(* IEC 61131-3 sources: com.logicals.lc3.examples/TF_Training/src/Blocks/Motor/FBD, 3 files *)

(* ---- FB_Motor1D_FBD.iecfbd ---- *)
FUNCTION_BLOCK FB_Motor1D_FBD
  VAR
    FB_MotorRS : RS;
    FB_MotorR_TRIG : R_TRIG;
    FB_MotorTON : TON;
  END_VAR
  VAR_INPUT
    vix_Start : BOOL;
    vix_Stop : BOOL;
  END_VAR
  VAR_OUTPUT
    vox_MotorOut : BOOL;
    vox_Err : BOOL;
    vox_ErrNo : INT;
  END_VAR

  (*

    // Network 1:
    FB_MotorR_TRIG(CLK := vix_Start);
    FB_MotorRS(S := FB_MotorR_TRIG.Q, R1 := vix_Stop, Q1 => vox_MotorOut);

    // Network 2:
    AND(IN1 := vix_Start, IN2 := vix_Stop, AND => vox_Err);

    // Network 3:
    AND(IN1 := vix_Start, IN2 := vix_Stop, AND => @C(19).AND);
    MOVE(EN := @C(19).AND, IN := 1, MOVE => vox_ErrNo);

  *)

  @CF(11) : @R(620.0, 130.0, 670.0, 39.0), @T("Motor_1D"), @POU;
  @VF(1) : @E(vix_Start), @R(620.0, 210.0, 140.0, 19.0);
  @VF(2) : @E(vix_Stop), @R(620.0, 260.0, 140.0, 19.0);
  @C(3) : @FB(FB_MotorR_TRIG), @R(840.0, 210.0, 140.0, 18.0), @I(@N(CLK), @L(9.5)), @O(@N(Q), @R(9.5));
  @C(4) : @FB(FB_MotorRS), @R(1030.0, 210.0, 80.0, 38.0), @I(@N(S), @L(9.5)), @I(@N(R1), @L(29.5)), @O(@N(Q1), @R(9.5));
  @VF(8) : @E(vox_MotorOut), @R(1150.0, 210.0, 140.0, 19.0);
  @CF(10) : @R(620.0, 330.0, 670.0, 39.0), @T("Motor_1D - Error Bit"), @POU;
  @VF(12) : @E(vix_Start), @R(620.0, 400.0, 140.0, 19.0);
  @VF(13) : @E(vix_Stop), @R(620.0, 420.0, 140.0, 19.0);
  @C(14) : @F(AND), @R(860.0, 400.0, 40.0, 38.0), BOOL, @I(@N(IN1), @L(9.5)), @I(@N(IN2), @L(29.5)), @O(@N(AND), @R(9.5));
  @VF(17) : @E(vox_Err), @R(1150.0, 400.0, 140.0, 19.0);
  @C(19) : @F(AND), @R(860.0, 560.0, 40.0, 38.0), BOOL, @I(@N(IN1), @L(9.5)), @I(@N(IN2), @L(29.5)), @O(@N(AND), @R(9.5));
  @VF(20) : @E(vix_Start), @R(620.0, 560.0, 140.0, 19.0);
  @VF(21) : @E(vix_Stop), @R(620.0, 580.0, 140.0, 19.0);
  @VF(22) : @E(vox_ErrNo), @R(1150.0, 580.0, 140.0, 19.0);
  @CF(23) : @R(620.0, 490.0, 670.0, 39.0), @T("Motor_1D - Error No"), @POU;
  @C(26) : @F(MOVE), @R(1000.0, 560.0, 60.0, 38.0), INT, @I(@N(EN), @L(9.5)), @I(@N(IN), @L(29.5)), @O(@N(ENO), @R(9.5)), @O(@N(MOVE), @R(29.5));
  @VF(29) : @E(1), @R(760.0, 620.0, 140.0, 19.0), INT;
  @OLT(31) : @R(1360.0, 210.0, 80.0, 19.0), @S(8);

  @G(5) :
     @L(@VF(1).o, @C(3).CLK)
    ;
  @G(6) :
     @L(@C(3).Q, @C(4).S)
    ;
  @G(7) :
     @L(@VF(2).o, @C(4).R1)
    ;
  @G(9) :
     @L(@C(4).Q1, @VF(8).i)
    ;
  @G(15) :
     @L(@VF(12).o, @C(14).IN1)
    ;
  @G(16) :
     @L(@VF(13).o, @C(14).IN2)
    ;
  @G(18) :
     @L(@C(14).AND, @VF(17).i)
    ;
  @G(24) :
     @L(@VF(20).o, @C(19).IN1)
    ;
  @G(25) :
     @L(@VF(21).o, @C(19).IN2)
    ;
  @G(27) :
     @L(@C(19).AND, @C(26).EN)
    ;
  @G(28) :
     @L(@C(26).MOVE, @VF(22).i)
    ;
  @G(30) :
     @L(@VF(29).o, @C(26).IN)
    ;
END_FUNCTION_BLOCK

(* ---- FB_Motor2D_FBD.iecfbd ---- *)
FUNCTION_BLOCK FB_Motor2D_FBD
  {
    width := 310;
  }

  VAR
    FB_LeftRS : RS;
    FB_RightRS : RS;
    FB_LeftR_TRIG : R_TRIG;
    FB_RightR_TRIG : R_TRIG;
    FB_LeftTON : TON;
    FB_RightTON : TON;
  END_VAR
  VAR
    lx_LeftPulse : BOOL;
    lx_RightPulse : BOOL;
  END_VAR
  VAR_INPUT
    vix_Left : BOOL;
    vix_Right : BOOL;
    vix_LeftFB : BOOL;
    vix_RightFB : BOOL;
    vit_LeftFBTime : TIME := T#10m;
    vit_RightFBTime : TIME := T#10m;
  END_VAR
  VAR_OUTPUT
    vox_MotorLeft : BOOL;
    vox_MotorRight : BOOL;
    vox_LeftFBErr : BOOL;
    vox_RightFBErr : BOOL;
    vox_Err : BOOL;
    vox_ErrNo : INT;
  END_VAR

  (*

    // Network 1:
    FB_RightR_TRIG(CLK := vix_Right, Q => lx_RightPulse);

    // Network 2:
    FB_LeftR_TRIG(CLK := vix_Left, Q => lx_LeftPulse);

    // Network 3:
    AND(IN1 := vix_Left, IN2 := vix_Right, AND => vox_Err);

    // Network 4:
    AND(IN1 := vix_Left, IN2 := vix_Right, AND => @C(39).AND);
    MOVE(EN := @C(39).AND, IN := 1, MOVE => vox_ErrNo);

    // Network 5:
    FB_RightRS(S := lx_RightPulse, R1 := vox_MotorLeft, Q1 => vox_MotorRight);

    // Network 6:
    FB_LeftRS(S := lx_LeftPulse, R1 := vox_MotorRight, Q1 => vox_MotorLeft);

  *)

  @C(1) : @FB(FB_RightR_TRIG), @R(910.0, 150.0, 140.0, 18.0), @I(@N(CLK), @L(9.5)), @O(@N(Q), @R(9.5));
  @C(2) : @FB(FB_LeftR_TRIG), @R(910.0, 250.0, 140.0, 18.0), @I(@N(CLK), @L(9.5)), @O(@N(Q), @R(9.5));
  @VF(3) : @E(lx_LeftPulse), @R(1180.0, 250.0, 140.0, 19.0);
  @VF(4) : @E(lx_RightPulse), @R(1180.0, 150.0, 140.0, 19.0);
  @VF(7) : @E(vix_Left), @R(650.0, 250.0, 140.0, 19.0);
  @VF(9) : @E(vix_Right), @R(650.0, 150.0, 140.0, 19.0);
  @CF(11) : @R(650.0, 90.0, 670.0, 39.0), @T("Right R_TRIG"), @POU;
  @CF(12) : @R(650.0, 190.0, 670.0, 39.0), @T("Left R_TRIG"), @POU;
  @C(13) : @FB(FB_LeftRS), @R(990.0, 520.0, 80.0, 38.0), @I(@N(S), @L(9.5)), @I(@N(R1), @L(29.5)), @O(@N(Q1), @R(9.5));
  @C(14) : @FB(FB_RightRS), @R(990.0, 400.0, 80.0, 38.0), @I(@N(S), @L(9.5)), @I(@N(R1), @L(29.5)), @O(@N(Q1), @R(9.5));
  @VF(15) : @E(lx_RightPulse), @R(650.0, 400.0, 140.0, 19.0);
  @VF(17) : @E(lx_LeftPulse), @R(650.0, 520.0, 140.0, 19.0);
  @VF(19) : @E(vox_MotorLeft), @R(1180.0, 520.0, 140.0, 19.0);
  @VF(21) : @E(vox_MotorRight), @R(1180.0, 400.0, 140.0, 19.0);
  @CF(23) : @R(650.0, 330.0, 670.0, 39.0), @T("Left turn"), @POU;
  @CF(24) : @R(650.0, 460.0, 670.0, 39.0), @T("Right turn"), @POU;
  @VF(25) : @E(vox_MotorLeft), @R(650.0, 420.0, 140.0, 19.0);
  @VF(27) : @E(vox_MotorRight), @R(650.0, 540.0, 140.0, 19.0);
  @CF(29) : @R(650.0, 640.0, 680.0, 39.0), @T("Error bit"), @POU;
  @VF(30) : @E(vox_Err), @R(1190.0, 700.0, 140.0, 19.0);
  @VF(31) : @E(vix_Left), @R(660.0, 700.0, 140.0, 19.0);
  @VF(32) : @E(vix_Right), @R(660.0, 720.0, 140.0, 19.0);
  @C(33) : @F(AND), @R(1000.0, 700.0, 40.0, 38.0), BOOL, @I(@N(IN1), @L(9.5)), @I(@N(IN2), @L(29.5)), @O(@N(AND), @R(9.5));
  @CF(37) : @R(650.0, 780.0, 680.0, 39.0), @T("Error no"), @POU;
  @VF(38) : @E(vox_ErrNo), @R(1190.0, 880.0, 140.0, 19.0);
  @C(39) : @F(AND), @R(970.0, 860.0, 40.0, 38.0), BOOL, @I(@N(IN1), @L(9.5)), @I(@N(IN2), @L(29.5)), @O(@N(AND), @R(9.5));
  @VF(40) : @E(vix_Left), @R(660.0, 860.0, 140.0, 19.0);
  @VF(41) : @E(vix_Right), @R(660.0, 880.0, 140.0, 19.0);
  @C(44) : @F(MOVE), @R(1100.0, 860.0, 60.0, 38.0), INT, @I(@N(EN), @L(9.5)), @I(@N(IN), @L(29.5)), @O(@N(ENO), @R(9.5)), @O(@N(MOVE), @R(29.5));
  @VF(47) : @E(1), @R(870.0, 910.0, 140.0, 19.0), INT;
  @CF(49) : @R(650.0, 980.0, 680.0, 39.0), @T("Delay FB not used up to now!"), @POU;

  @G(5) :
     @L(@C(1).Q, @VF(4).i)
    ;
  @G(6) :
     @L(@C(2).Q, @VF(3).i)
    ;
  @G(8) :
     @L(@VF(7).o, @C(2).CLK)
    ;
  @G(10) :
     @L(@VF(9).o, @C(1).CLK)
    ;
  @G(16) :
     @L(@VF(15).o, @C(14).S)
    ;
  @G(18) :
     @L(@VF(17).o, @C(13).S)
    ;
  @G(20) :
     @L(@C(13).Q1, @VF(19).i)
    ;
  @G(22) :
     @L(@C(14).Q1, @VF(21).i)
    ;
  @G(26) :
     @L(@VF(25).o, @C(14).R1)
    ;
  @G(28) :
     @L(@VF(27).o, @C(13).R1)
    ;
  @G(34) :
     @L(@VF(31).o, @C(33).IN1)
    ;
  @G(35) :
     @L(@VF(32).o, @C(33).IN2)
    ;
  @G(36) :
     @L(@C(33).AND, @VF(30).i)
    ;
  @G(42) :
     @L(@VF(40).o, @C(39).IN1)
    ;
  @G(43) :
     @L(@VF(41).o, @C(39).IN2)
    ;
  @G(45) :
     @L(@C(44).MOVE, @VF(38).i)
    ;
  @G(46) :
     @L(@C(39).AND, @C(44).EN)
    ;
  @G(48) :
     @L(@VF(47).o, @C(44).IN)
    ;
END_FUNCTION_BLOCK

(* ---- FB_Motor2D_STOP_FBD.iecfbd ---- *)
FUNCTION_BLOCK FB_Motor2D_STOP_FBD
  {
    width := 380;
  }

  VAR
    FB_LeftRS : RS;
    FB_RightRS : RS;
    FB_LeftR_TRIG : R_TRIG;
    FB_RightR_TRIG : R_TRIG;
    FB_LeftTON : TON;
    FB_RightTON : TON;
    FB_RightR_TRIG1 : R_TRIG;
    FB_LeftR_TRIG1 : R_TRIG;
    FB_RightRS1 : RS;
    FB_LeftRS1 : RS;
  END_VAR
  VAR
    lx_LeftPulse : BOOL;
    lx_RightPulse : BOOL;
  END_VAR
  VAR_INPUT
    vix_Left : BOOL;
    vix_Right : BOOL;
    vix_Stop : BOOL;
    vix_LeftFB : BOOL;
    vix_RightFB : BOOL;
    vix_MotorProt : BOOL;
    vit_LeftFBTime : TIME := T#10m;
    vit_RightFBTime : TIME := T#10m;
  END_VAR
  VAR_OUTPUT
    vox_MotorLeft : BOOL;
    vox_MotorRight : BOOL;
    vox_LeftFBErr : BOOL;
    vox_RightFBErr : BOOL;
    vix_MotorProtErr : BOOL;
    vox_Err : BOOL;
    vox_ErrNo : INT;
  END_VAR

  (*

    // Network 1:
    FB_RightR_TRIG1(CLK := vix_Right, Q => lx_RightPulse);

    // Network 2:
    FB_LeftR_TRIG1(CLK := vix_Left, Q => lx_LeftPulse);

    // Network 3:
    NOT(IN := vox_MotorLeft, NOT => @C(54).NOT);
    AND(IN1 := lx_LeftPulse, IN2 := @C(54).NOT, AND => @C(57).AND);
    FB_LeftRS1(S := @C(57).AND, R1 := vix_Stop, Q1 => vox_MotorLeft);

    // Network 4:
    NOT(IN := vox_MotorLeft, NOT => @C(51).NOT);
    AND(IN1 := lx_RightPulse, IN2 := @C(51).NOT, AND => @C(49).AND);
    FB_RightRS1(S := @C(49).AND, R1 := vix_Stop, Q1 => vox_MotorRight);

    // Network 5:
    AND(IN1 := vix_Left, IN2 := vix_Right, AND => vox_Err);

    // Network 6:
    AND(IN1 := vix_Left, IN2 := vix_Right, AND => @C(39).AND);
    MOVE(EN := @C(39).AND, IN := 1, MOVE => vox_ErrNo);

  *)

  @C(1) : @FB(FB_RightR_TRIG1), @R(780.0, 130.0, 140.0, 18.0), @I(@N(CLK), @L(9.5)), @O(@N(Q), @R(9.5));
  @C(2) : @FB(FB_LeftR_TRIG1), @R(780.0, 230.0, 140.0, 18.0), @I(@N(CLK), @L(9.5)), @O(@N(Q), @R(9.5));
  @C(14) : @FB(FB_RightRS1), @R(860.0, 380.0, 80.0, 38.0), @I(@N(S), @L(9.5)), @I(@N(R1), @L(29.5)), @O(@N(Q1), @R(9.5));
  @C(13) : @FB(FB_LeftRS1), @R(860.0, 600.0, 80.0, 38.0), @I(@N(S), @L(9.5)), @I(@N(R1), @L(29.5)), @O(@N(Q1), @R(9.5));
  @C(33) : @F(AND), @R(870.0, 820.0, 40.0, 38.0), BOOL, @I(@N(IN1), @L(9.5)), @I(@N(IN2), @L(29.5)), @O(@N(AND), @R(9.5));
  @C(39) : @F(AND), @R(840.0, 980.0, 40.0, 38.0), BOOL, @I(@N(IN1), @L(9.5)), @I(@N(IN2), @L(29.5)), @O(@N(AND), @R(9.5));
  @C(44) : @F(MOVE), @R(970.0, 980.0, 60.0, 38.0), INT, @I(@N(EN), @L(9.5)), @I(@N(IN), @L(29.5)), @O(@N(ENO), @R(9.5)), @O(@N(MOVE), @R(29.5));
  @VF(9) : @E(vix_Right), @R(520.0, 130.0, 140.0, 19.0);
  @VF(7) : @E(vix_Left), @R(520.0, 230.0, 140.0, 19.0);
  @VF(15) : @E(lx_RightPulse), @R(520.0, 380.0, 140.0, 19.0);
  @VF(25) : @E(vox_MotorLeft), @R(520.0, 400.0, 140.0, 19.0);
  @VF(3) : @E(lx_LeftPulse), @R(1050.0, 230.0, 140.0, 19.0);
  @VF(4) : @E(lx_RightPulse), @R(1050.0, 130.0, 140.0, 19.0);
  @VF(21) : @E(vox_MotorRight), @R(1050.0, 380.0, 140.0, 19.0);
  @VF(17) : @E(lx_LeftPulse), @R(520.0, 600.0, 140.0, 19.0);
  @VF(19) : @E(vox_MotorLeft), @R(1050.0, 600.0, 140.0, 19.0);
  @VF(31) : @E(vix_Left), @R(520.0, 820.0, 140.0, 19.0);
  @VF(30) : @E(vox_Err), @R(1060.0, 820.0, 140.0, 19.0);
  @VF(32) : @E(vix_Right), @R(520.0, 840.0, 140.0, 19.0);
  @VF(38) : @E(vox_ErrNo), @R(1060.0, 1000.0, 140.0, 19.0);
  @VF(40) : @E(vix_Left), @R(520.0, 980.0, 140.0, 19.0);
  @VF(41) : @E(vix_Right), @R(520.0, 1000.0, 140.0, 19.0);
  @VF(47) : @E(1), @R(740.0, 1030.0, 140.0, 19.0), INT;
  @CF(11) : @R(520.0, 70.0, 670.0, 39.0), @T("Right R_TRIG"), @POU;
  @CF(12) : @R(520.0, 170.0, 670.0, 39.0), @T("Left R_TRIG"), @POU;
  @CF(23) : @R(520.0, 310.0, 670.0, 39.0), @T("Right turn"), @POU;
  @CF(24) : @R(520.0, 540.0, 670.0, 39.0), @T("Left turn"), @POU;
  @CF(29) : @R(520.0, 760.0, 680.0, 39.0), @T("Error bit"), @POU;
  @CF(37) : @R(520.0, 900.0, 680.0, 39.0), @T("Error no"), @POU;
  @VF(26) : @E(vix_Stop), @R(520.0, 450.0, 140.0, 19.0);
  @C(49) : @F(AND), @R(770.0, 380.0, 40.0, 38.0), BOOL, @I(@N(IN1), @L(9.5)), @I(@N(IN2), @L(29.5)), @O(@N(AND), @R(9.5));
  @C(51) : @F(NOT), @R(690.0, 400.0, 60.0, 18.0), BOOL, @I(@N(IN), @L(9.5)), @O(@N(NOT), @R(9.5));
  @C(54) : @F(NOT), @R(690.0, 620.0, 60.0, 18.0), BOOL, @I(@N(IN), @L(9.5)), @O(@N(NOT), @R(9.5));
  @VF(55) : @E(vox_MotorLeft), @R(520.0, 620.0, 140.0, 19.0);
  @C(57) : @F(AND), @R(780.0, 600.0, 40.0, 38.0), BOOL, @I(@N(IN1), @L(9.5)), @I(@N(IN2), @L(29.5)), @O(@N(AND), @R(9.5));
  @VF(61) : @E(vix_Stop), @R(520.0, 680.0, 140.0, 19.0);
  @CF(28) : @R(520.0, 1150.0, 670.0, 39.0), @T("Delay FB not used up to now!"), @POU;

  @G(10) :
     @L(@VF(9).o, @C(1).CLK)
    ;
  @G(8) :
     @L(@VF(7).o, @C(2).CLK)
    ;
  @G(5) :
     @L(@C(1).Q, @VF(4).i)
    ;
  @G(6) :
     @L(@C(2).Q, @VF(3).i)
    ;
  @G(16) :
     @L(@VF(15).o, @C(49).IN1)
    ;
  @G(22) :
     @L(@C(14).Q1, @VF(21).i)
    ;
  @G(20) :
     @L(@C(13).Q1, @VF(19).i)
    ;
  @G(34) :
     @L(@VF(31).o, @C(33).IN1)
    ;
  @G(36) :
     @L(@C(33).AND, @VF(30).i)
    ;
  @G(35) :
     @L(@VF(32).o, @C(33).IN2)
    ;
  @G(42) :
     @L(@VF(40).o, @C(39).IN1)
    ;
  @G(46) :
     @L(@C(39).AND, @C(44).EN)
    ;
  @G(43) :
     @L(@VF(41).o, @C(39).IN2)
    ;
  @G(45) :
     @L(@C(44).MOVE, @VF(38).i)
    ;
  @G(48) :
     @L(@VF(47).o, @C(44).IN)
    ;
  @G(50) :
     @L(@C(49).AND, @C(14).S)
    ;
  @G(52) :
     @L(@VF(25).o, @C(51).IN)
    ;
  @G(53) :
     @L(@C(51).NOT, @C(49).IN2)
    ;
  @G(56) :
     @L(@VF(55).o, @C(54).IN)
    ;
  @G(18) :
     @L(@VF(17).o, @C(57).IN1)
    ;
  @G(58) :
     @L(@C(57).AND, @C(13).S)
    ;
  @G(59) :
     @L(@VF(26).o, @C(14).R1)
    ;
  @G(60) :
     @L(@C(54).NOT, @C(57).IN2)
    ;
  @G(27) :
     @L(@VF(61).o, @C(13).R1)
    ;
END_FUNCTION_BLOCK
